Staubli VAL3: Bool_Edit.pgx

public program Bool_Edit(bool& x_bRes, num x_nX, num x_nY, num x_nLength)
  local num l_nNum
  local string l_s[2]
begin

//在下拉选择框中
//是否选择

  l_s[1]="是"
  l_s[0]="否"


   call BoolMess_Edit(x_bRes,x_nX,x_nY,x_nLength,l_s)

end
